FUNCTION_BLOCK FB_SerialComPort_Base
VAR_INPUT
END_VAR
VAR_OUTPUT
	bIsWorking 	: BOOL;
	bIsLocked	: BOOL;
END_VAR
VAR
	RxBufferSerialCom  	: Tc2_SerialCom.ComBuffer;
	TxBufferSerialCom  	: Tc2_SerialCom.ComBuffer;
	fbClearComBuffer	: Tc2_SerialCom.ClearComBuffer;
	fbFifo				: FB_SimpleFIFO_PVOID;
	bLock				: BOOL;
	rTrig				: R_TRIG;
	timerLock			: TON;
END_VAR

timerLock();
IF timerLock.Q THEN
	timerLock(IN:= FALSE);
	bIsLocked := FALSE;
END_IF

METHOD M_ClearRxComBuffer
VAR_INPUT
END_VAR
fbClearComBuffer(buffer := RxBufferSerialCom);
END_METHOD

METHOD M_ClearTxComBuffer
VAR_INPUT
END_VAR
fbClearComBuffer(buffer := TxBufferSerialCom);
END_METHOD

METHOD M_IsMyTurn : BOOL
VAR_INPUT
	pInstance : PVOID;
END_VAR
M_IsMyTurn := fbFifo.M_GetHead() = pInstance;
END_METHOD

METHOD M_LockForTime
VAR_INPUT
	tLockTime : TIME;
END_VAR
timerLock.IN := TRUE;
timerLock.PT := tLockTime;
bIsLocked := TRUE;
END_METHOD

METHOD M_Register : BOOL
VAR_INPUT
	pInstance : PVOID;
END_VAR
M_Register := fbFifo.M_Add(pInstance);
END_METHOD

METHOD M_Release : BOOL
VAR_INPUT
	pInstance : PVOID;
END_VAR
M_Release := fbFifo.M_Remove(pInstance);
END_METHOD

PROPERTY P_RxBuffer : REFERENCE TO Tc2_SerialCom.ComBuffer
GET
P_RxBuffer REF= RxBufferSerialCom;
END_GET
END_PROPERTY

PROPERTY P_TxBuffer : REFERENCE TO Tc2_SerialCom.ComBuffer
GET
P_TxBuffer REF= TxBufferSerialCom;
END_GET
END_PROPERTY

END_FUNCTION_BLOCK

(* stored: Version 1.1.0.1, ProductVersion 3.1.4024.6
   POU FB_SerialComPort_Base: Id {dafc142e-3448-4161-a494-645e6b6fc2b9}, SpecialFunc None
   Method M_ClearRxComBuffer: Id {332aa9fb-e536-4b99-a85f-5f887b31edb5}
   Method M_ClearTxComBuffer: Id {1bec5137-ba4d-4171-ada5-e7038643fefd}
   Method M_IsMyTurn: Id {baa7b5fa-53e6-41d1-9e2f-d5fc2a2148f1}
   Method M_LockForTime: Id {898bd436-bc77-4d73-a421-e307320706b2}
   Method M_Register: Id {c68d76a8-c588-49a6-8626-9c21c307f594}
   Method M_Release: Id {723d8d7d-b271-4973-bef0-c2097d6eca8a}
   Property P_RxBuffer: Id {b535b9fd-49c7-40c8-869a-6dde081406d4}
   Get Get: Id {ea137d5e-601f-47c2-abcd-3f046e772675}
   Property P_TxBuffer: Id {53a2f75f-34bd-4aec-b1d3-b1b4202d4aa3}
   Get Get: Id {86315931-b7f4-42fc-afa9-e043df95388e} *)
